(* PLC project 117_1_V0.5.project, CODESYS CODESYS V3.5 SP17 Patch 3 *)
(* stored: creationDateTime 1970-01-01T00:00:00, modificationDateTime 2026-06-16T22:51:19.9979415 *)

(* values of PID_DIRECTION_UDT: DIRECT: [0] Прямая работа: ошибка = SP - PV; REVERSE: [1] Обратная работа: ошибка = PV - SP *)

{attribute 'strict'}
TYPE PID_DIRECTION_UDT : (DIRECT, REVERSE);
END_TYPE
